FUNCTION_BLOCK Case
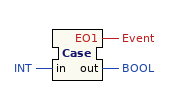
  EVENT_OUTPUT
    EO1;
  END_EVENT
  VAR_INPUT
    in : INT;
  END_VAR
  VAR_OUTPUT
    out : BOOL;
  END_VAR
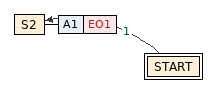
  EC_STATES
    START;
    S2 : A1 -> EO1;
  END_STATES
  EC_TRANSITIONS
    START TO S2 := 1;
  END_TRANSITIONS
  ALGORITHM A1 IN ST:
CASE in OF &#38;#10;  0 -&#62;&#38;#10;    out := FALSE;&#38;#10;  1 -&#62;&#38;#10;    out := TRUE;&#38;#10;  2 -&#62;&#38;#10;    out := TRUE;&#38;#10;  TRUE -&#62;&#38;#10;    out := FALSE;&#38;#10;END_CASE;&#38;#10;
  END_ALGORITHM
END_FUNCTION_BLOCK
